{attribute addProperty BoxType "KL3361"}
{attribute addProperty Id "Channel_1Channel_D054A87F00"}
{attribute addProperty CRC "2211813723"}
{attribute addProperty SizeInBites "0"}
{attribute addProperty SizeInBytes "0"}
TYPE KL3361_83D5995B :
STRUCT
	{attribute addProperty Name "Channel_1"}
	Channel_1 : Channel_D054A87F;
END_STRUCT
END_TYPE

(* stored: Version 1.2.0.0, ProductVersion 3.1.4024.9
   DUT KL3361_83D5995B: Id {32edc01b-8d93-4806-b263-b24d52f67e6e} *)
